// Brief: Master Arm Error Hold
FUNCTION_BLOCK PUBLIC FB_StateCtrlError EXTENDS FB_SlaveArmCtrlBase
VAR_INPUT
END_VAR
VAR_OUTPUT
END_VAR
VAR
END_VAR

// override this function in each exact controller
// NOTICE: set joint control mode here, and do some initialization if needed
METHOD PUBLIC init : BOOL
VAR_IN_OUT CONSTANT
	i_slaveArm	:FB_SlaveArm;
END_VAR
VAR_IN_OUT 
	r_slaveArmCtrlCmd :ST_SlaveArmCtrlCmds;
END_VAR


VAR
	i:INT;
END_VAR
SUPER^.Init(i_slaveArm,r_slaveArmCtrlCmd);

// disable all joints
 m_jntEnableFlag :=g_zeroVec8i;
END_METHOD

END_FUNCTION_BLOCK

(* stored: Version 1.1.0.1, ProductVersion 3.1.4024.12
   POU FB_StateCtrlError: Id {78b2e60d-537e-446e-8b3b-6db63d5ab02c}, SpecialFunc None
   Method init: Id {e6a6f329-eae4-4e64-b8ba-0dd027b37a8e} *)
